(* FB_Cylinder		- number of control signals:
							one direction is controllable
					- type of feedback signal:
							feedback in base and work position		*)
						
FUNCTION_BLOCK FB_Cylinder
VAR_INPUT
	bAtBasePos		AT %I*	: BOOL;		// Hardware input signal: cylinder is at base position
	bAtWorkPos		AT %I*	: BOOL;		// Hardware input signal: cylinder is at work position
END_VAR
VAR_OUTPUT
	bMoveToWork		AT %Q*	: BOOL;		// Hardware output signal to move cylinder to work position
	bMoveToBase		AT %Q*	: BOOL;		// Hardware output signal to move cylinder to base position
END_VAR

// =========================================================
;
// =========================================================

PROPERTY PUBLIC bState_AtBasePos : BOOL
GET
bState_AtBasePos := bAtBasePos;
END_GET
END_PROPERTY

PROPERTY PUBLIC bState_AtWorkPos : BOOL
GET
bState_AtWorkPos := bAtWorkPos;
END_GET
END_PROPERTY

PROPERTY bState_MoveToBase : bool
GET
bState_MoveToBase := bMoveToBase;
END_GET
END_PROPERTY

PROPERTY PUBLIC bState_MoveToWork : BOOL
GET
bState_MoveToWork := bMoveToWork;
END_GET
END_PROPERTY

METHOD MoveToBase
VAR_INPUT
END_VAR
// =========================================================
	
StateMachine(	bBasePosReq := TRUE,
				bWorkPosReq	:= FALSE );
							
// =========================================================
END_METHOD

METHOD MoveToWork
VAR_INPUT
END_VAR
// =========================================================
	
StateMachine(	bBasePosReq := FALSE,
				bWorkPosReq	:= TRUE );
								
// =========================================================
END_METHOD

METHOD Reset
VAR_INPUT
END_VAR
// =========================================================

bMoveToWork := FALSE;
bMoveToBase	:= TRUE;

// =========================================================
END_METHOD

METHOD PROTECTED StateMachine
VAR_INPUT
	bBasePosReq		: BOOL;
	bWorkPosReq		: BOOL;
END_VAR
// =========================================================
// Base or work position requested
		
	IF bWorkPosReq THEN
		bMoveToWork := TRUE;
		bMoveToBase	:= FALSE;
	END_IF
	
	IF bBasePosReq THEN
		bMoveToWork := FALSE;
		bMoveToBase	:= TRUE;
	END_IF

// =========================================================
END_METHOD

END_FUNCTION_BLOCK

(* stored: Version 1.1.0.1, ProductVersion 3.1.4024.12
   POU FB_Cylinder: Id {049cf0c8-787e-48cd-9dba-779e7bf86b9c}, SpecialFunc None
   Property bState_AtBasePos: Id {c0b0975a-26f1-4b20-88a5-afa52a3876df}
   Get Get: Id {f0bf4a4f-2389-4d61-bdc9-c73a151c3463}
   Property bState_AtWorkPos: Id {50b0f44d-9561-4544-8a01-7e892601d662}
   Get Get: Id {8d8443a6-9502-4ef4-bee9-85be4bb5027b}
   Property bState_MoveToBase: Id {77dc67ca-ba1e-4826-93fe-38cd9412a291}
   Get Get: Id {5c2332e8-bf14-4055-b910-719395e6d125}
   Property bState_MoveToWork: Id {6e781349-f89a-4e7b-9cf8-53327ab40deb}
   Get Get: Id {1b73982c-b6aa-4870-aa30-8ad51a8d202c}
   Method MoveToBase: Id {1bd60d0a-72f1-4adb-a81d-66a2f8af9c07}
   Method MoveToWork: Id {9657ee8e-90c8-45ee-8d0d-3c02ce9d1ba2}
   Method Reset: Id {ffd7021d-b698-4257-8d7a-ae703597054a}
   Method StateMachine: Id {c854d137-c5dd-4da4-bf25-36bb7c20932d} *)
